// TIA Portal V18 export
DATA_BLOCK "SS2_A2_8AO_AO_Vars"   // DB11131
{ S7_Optimized_Access := 'FALSE' }
VERSION : 0.1
// stored: AutoNumber false, DBAccessibleFromOPCUA true, IsOnlyStoredInLoadMemory false, IsWriteProtectedInAS false
   VAR
      AO1 { S7_SetPoint := 'True'} : "UDT_AOadv";
      AO2 { S7_SetPoint := 'True'} : "UDT_AOadv";
      AO3 : "UDT_AOadv";
      AO4 : "UDT_AOadv";
      AO5 { S7_SetPoint := 'True'} : "UDT_AOadv";
      AO6 { S7_SetPoint := 'True'} : "UDT_AOadv";
      AO7 { S7_SetPoint := 'True'} : "UDT_AOadv";
      AO8 { S7_SetPoint := 'True'} : "UDT_AOadv";
   END_VAR
BEGIN
   AO1.cMOA := 1;
   AO1.cFuncSystemID := 2;
   AO1.cFuncVar := 2;
   AO1.rManOutput := 100.0;
   AO2.cFuncSystemID := 2;
   AO2.cFuncVar := 3;
END_DATA_BLOCK
